FUNCTION Convert_UDINT_TO_WORD : Hresult
VAR_INPUT
	in : UDINT;
	out : REFERENCE TO WORD;
END_VAR
VAR
	converted : WORD;
END_VAR
VAR CONSTANT
	INCOMPATIBLE : HRESULT := 16#9811070E;
END_VAR

converted := UDINT_TO_WORD(in);

IF (WORD_TO_UDINT(converted) <> in) THEN
	Convert_UDINT_TO_WORD := INCOMPATIBLE;
	RETURN;
END_IF

out := converted;

END_FUNCTION

(* stored: Version 1.1.0.1, ProductVersion 3.1.4024.12
   POU Convert_UDINT_TO_WORD: Id {d0269e1e-aaa0-43ed-b0e0-4da498e51428}, SpecialFunc None *)
